Fanuc KAREL source: ka00092.KL

-- PROVISIONAL review KL for V770-1; original PC SHA256 82ef1be9044b9e4880bee497062a4a594265a70f0a7020f039e92c0c4afab887
-- Incomplete behavior may be omitted. Consult companion uncertainty JSON. Do not deploy.
PROGRAM KA00092
%NOLOCKGROUP
-- UNRESOLVED_DECL SRC type=000199
-- UNRESOLVED_DECL DST type=000199
BEGIN
  -- UNRESOLVED_PC offsets 5-20; opcodes 49,4A
  -- UNRESOLVED_PC offsets 25-29; opcodes 7F
END KA00092
